{attribute 'qualified_only'}
VAR_GLOBAL
	{attribute 'OPC.UA.DA' := '1'}
	bBit			: BOOL;
	{attribute	'OPC.UA.DA'	:= '1'}
	nSayi			: INT;
	{attribute	'OPC.UA.DA'	:= '1'}
	sMetin			: STRING;
END_VAR

(* stored: Version 1.1.0.1, ProductVersion 3.1.4024.6
   GVL OPC: Id {29972865-3f79-451d-bde3-cdba0f08ef26} *)
